FUNCTION_BLOCK FB_SplitRealToWords
////////////////// 
// Convert one REAL into  2 separate WORDS in Big Endian Encoding. 
//////////////////	
VAR_INPUT
	IN		: REAL ;				// Real input
	
END_VAR

VAR_OUTPUT
	OUT		: ARRAY[0..1]OF WORD;	// Word output array
	
END_VAR

OUT[1] := DWORD_TO_WORD(SHR(SHL(REAL_TO_DWORD(IN),16),16)) ; 	// Strong Word
OUT[0] := DWORD_TO_WORD(SHR(REAL_TO_DWORD(IN),16)); 			// Weak Word

END_FUNCTION_BLOCK

(* stored: Version 1.1.0.1, ProductVersion 3.1.4024.6
   POU FB_SplitRealToWords: Id {54876f84-9ff2-45b8-9d42-47f66fa12b9e}, SpecialFunc None *)
